(* CODESYS project FU_lwBitGetPart.xml

Project tree, tasks and I/O mapping:
  function FU_lwBitGetPart [ST]
*)

// FU_lwBitGetPart
//This function gets only the needed bits of a variable
// |**Version**|**Author**| **Date** |**Changes**
// | 1         | NSN      | 16-03-22 | Creation
FUNCTION FU_lwBitGetPart : LWORD
VAR_INPUT
	value			:LWORD;		//Variable to get value from
	amount			:BYTE;		//Amount of bits to change
	offset			:BYTE;		//Offset in variable to change bits at
END_VAR

FU_lwBitGetPart		:=		SHR(value,offset) AND GConstants.binaryMaskLWord[amount];

END_FUNCTION
